% RSLogix 500 project project 8.RSS, saved by version 8.30.00.16 %
PROJECT "UNTITLED"    % processor: Bul.1763 MicroLogix 1100 Series B %

PROGRAM FILES
  LAD 2 "MAIN"  2 rungs
  LAD 3 "IO"  1 rungs
  LAD 4 "CNTRL"  7 rungs

DATA FILES
  O0 OUTPUT  4 elements
  I1 INPUT  6 elements
  S2 STATUS  66 elements
  B3 BINARY  2 elements
  T4 TIMER  1 elements
  C5 COUNTER  1 elements
  R6 CONTROL  1 elements
  N7 INTEGER  7 elements
  F8 FLOAT  2 elements
  N9 CONSTANTS  4 elements

LADDER 2 "MAIN"
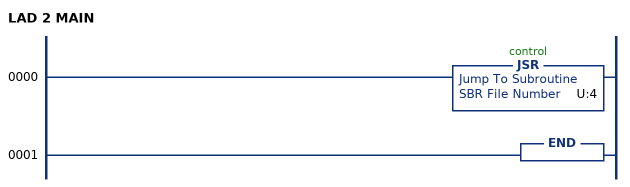
% Rung: 0 %
SOR JSR U:4 EOR
%   U:4  "control" %
% Rung: 1 %
SOR END EOR

LADDER 4 "CNTRL"
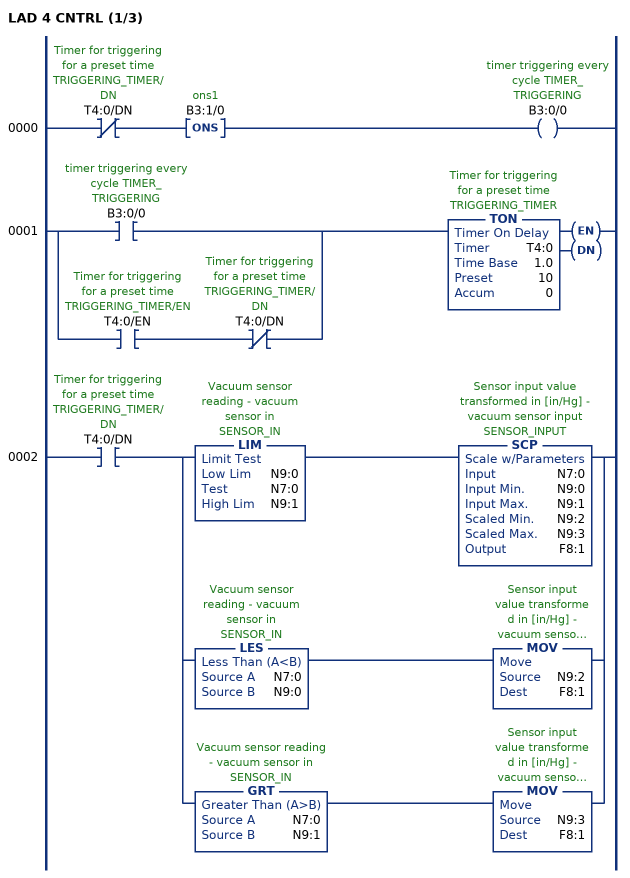
% Rung: 0 %
SOR XIO T4:0/DN ONS B3:1/0 OTE B3:0/0 EOR
%   T4:0  TRIGGERING_TIMER  "Timer for triggering for a preset time" %
%   B3:1/0  "ons1" %
%   B3:0/0  TIMER_TRIGGERING  "timer triggering every cycle" %
% Rung: 1 %
SOR BST XIC B3:0/0 NXB XIC T4:0/EN XIO T4:0/DN BND TON T4:0 1.0 10 0 EOR
%   B3:0/0  TIMER_TRIGGERING  "timer triggering every cycle" %
%   T4:0  TRIGGERING_TIMER  "Timer for triggering for a preset time" %
% Rung: 2 %
SOR XIC T4:0/DN BST LIM N9:0 N7:0 N9:1 SCP N7:0 N9:0 N9:1 N9:2 N9:3 F8:1 NXB LES N7:0 N9:0 MOV N9:2 F8:1 NXB GRT N7:0 N9:1 MOV N9:3 F8:1 BND EOR
%   T4:0  TRIGGERING_TIMER  "Timer for triggering for a preset time" %
%   N9:0  "Input vacuum sensor input [in bit scaling]" %
%   N7:0  SENSOR_IN  "Vacuum sensor reading - vacuum sensor in" %
%   N9:1  "Vacuum sensor in max [in bit scalling]" %
%   N9:2  "lowest sensor range end" %
%   N9:3  "highest sensor reading range end" %
%   F8:1  SENSOR_INPUT  "Sensor input value transformed in [in/Hg] - vacuum sensor input" %

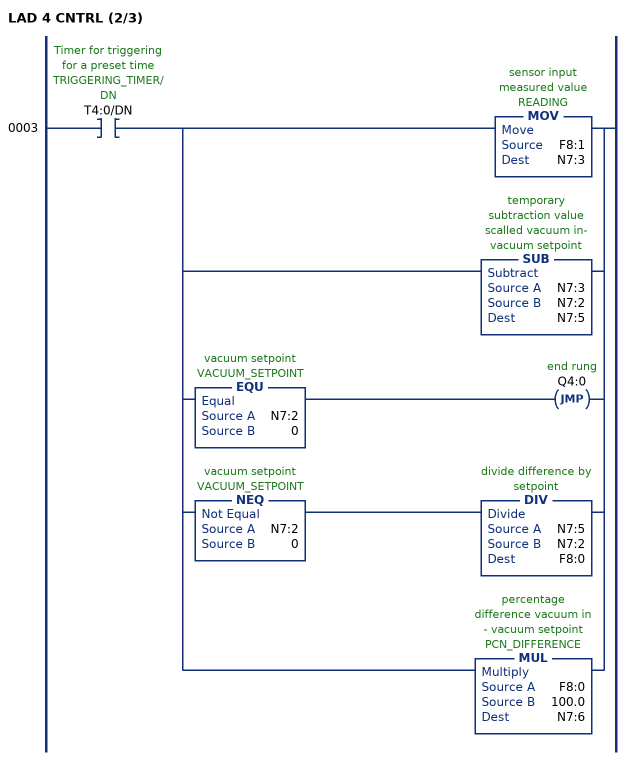
% Rung: 3 %
SOR XIC T4:0/DN BST MOV F8:1 N7:3 NXB SUB N7:3 N7:2 N7:5 NXB BST EQU N7:2 0 JMP Q4:0 NXB NEQ N7:2 0 DIV N7:5 N7:2 F8:0 BND NXB MUL F8:0 100.0 N7:6 BND EOR
%   T4:0  TRIGGERING_TIMER  "Timer for triggering for a preset time" %
%   F8:1  SENSOR_INPUT  "Sensor input value transformed in [in/Hg] - vacuum sensor input" %
%   N7:3  READING  "sensor input measured value" %
%   N7:2  VACUUM_SETPOINT  "vacuum setpoint" %
%   N7:5  "temporary subtraction value scalled vacuum in- vacuum setpoint" %
%   Q4:0  "end rung" %
%   F8:0  "divide difference by setpoint" %
%   N7:6  PCN_DIFFERENCE  "percentage difference vacuum in - vacuum setpoint" %

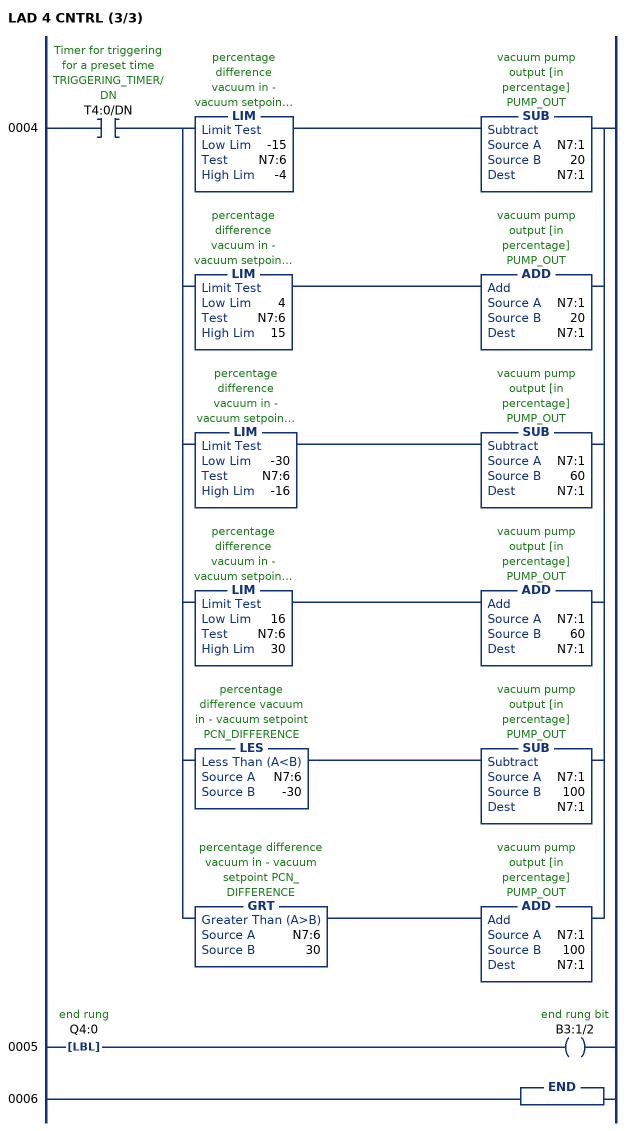
% Rung: 4 %
SOR XIC T4:0/DN BST LIM -15 N7:6 -4 SUB N7:1 20 N7:1 NXB LIM 4 N7:6 15 ADD N7:1 20 N7:1 NXB LIM -30 N7:6 -16 SUB N7:1 60 N7:1 NXB LIM 16 N7:6 30 ADD N7:1 60 N7:1 NXB LES N7:6 -30 SUB N7:1 100 N7:1 NXB GRT N7:6 30 ADD N7:1 100 N7:1 BND EOR
%   T4:0  TRIGGERING_TIMER  "Timer for triggering for a preset time" %
%   N7:6  PCN_DIFFERENCE  "percentage difference vacuum in - vacuum setpoint" %
%   N7:1  PUMP_OUT  "vacuum pump output [in percentage]" %
% Rung: 5 %
SOR LBL Q4:0 OTE B3:1/2 EOR
%   Q4:0  "end rung" %
%   B3:1/2  "end rung bit" %
% Rung: 6 %
SOR END EOR

OTHER DOCUMENTED ADDRESSES
  B3:1/1  "ons2"
  N7:4  "vacuum pump temporary value"

DATA TABLE (non-zero values as saved)
DATA T4
% .PRE .ACC %
% T4:0 % 10 0
DATA N9
% N9:0 % 0 16383 0 30
